//Placeholder, WIP --> need to define what purpose this struct serves
TYPE ST_SafetyStatus :
STRUCT
END_STRUCT
END_TYPE

(* stored: Version 1.1.0.1
   DUT ST_SafetyStatus: Id {00ac038e-aa81-4175-9c09-5cd4fbc6f3e8} *)
